KUKA KRL program: Wood_Test_2.src, Wood_Test_2.dat

--- Wood_Test_2.src ---
&ACCESS RVEO
&REL 38
&PARAM DISKPATH = KRC:\R1\Program\Milling
DEF Wood_Test_2 ( )
   INT lnActSt,lnUsedBase,lnActBase,lnUsedTool,lnBaseNr
   INT lnJobNr, lnCounter,lnCounter2
   FRAME lfZcut
   FRAME lfToolDiamShift
   FRAME lfStartMillingPos
   FRAME lfBaseShift
   FRAME lfBaseCycleZ
   FRAME lfBaseCycleShift

   CONTINUE
   ;IF ($T1 OR $T2)THEN
   GLOBAL INTERRUPT DECL 3 WHEN $STOPMESS==TRUE DO IR_STOPM ( )
   INTERRUPT ON 3
   BAS (#INITMOV,0)
   lnActSt = 1
   PTP $POS_ACT
   PTP lAstartPos

   gbRobControlActive = FALSE

   ; Used Base and tool
   lnUsedBase = 11
   lnActBase = 12
   lnUsedTool = 11

   gnLastToolNr = 5
   lnBaseNr = 23

   gfMillingOffset = $NULLFRAME

   lfZcut = $NULLFRAME
   lfZcut.Z = 0
   lfBaseShift = {X -30,Y -10,Z 1.1,A 0,B 0,C 0}
   lfBaseCycleZ = $NULLFRAME
   lfBaseCycleZ.Z = 0

   ;*************************************************************
   ;*                      Mill TOP SURFACE                     *
   ;*************************************************************
   grUsedRPM = GetMillingRPM(grTool_VC[gnLastToolNr], grTool_Diameter[gnLastToolNr])
   grUsedMillingSpeed = GetMillingSpeed(grUsedRPM, grTool_ToothCount[gnLastToolNr], grTool_FeedPerTooth[gnLastToolNr])

   SpindleRun(grUsedRPM,#CLOCKWISE)

   lfBaseCycleZ = $NULLFRAME
   lfBaseCycleZ.Z = 0
   BASE_DATA[lnUsedBase] = BASE_DATA[lnBaseNr] : lfBaseShift : lfBaseCycleZ
   TOOL_DATA[lnUsedTool] = TOOL_DATA[gnLastToolNr] :{X 0,Y 0,Z 0,A 270,B 0,C 0}

   MoveSettings(lnUsedBase, lnUsedTool, 100, grUsedMillingSpeed)
   ;; Move To PreposMillingPos Point P1 {5mm far from WP surface}
   lfToolDiamShift   = $NULLFRAME
   lfToolDiamShift.X = 0
   lfToolDiamShift.Y = 0
   lfToolDiamShift.Z = 5
   lfStartMillingPos = lfWorkPos[1] : lfToolDiamShift
   LIN lfStartMillingPos

   lfBaseCycleShift = $NULLFRAME
   BASE_DATA[lnActBase] = BASE_DATA[lnUsedBase]
   FOR lnCounter = 1 TO 2

      FOR lnCounter2 = 1 TO 2
         SWITCH lnCounter2
            CASE 1
               grUsedRPM = GetMillingRPM(grTool_VC[gnLastToolNr], grTool_Diameter[gnLastToolNr])
               grUsedMillingSpeed = GetMillingSpeed(grUsedRPM, grTool_ToothCount[gnLastToolNr], grTool_FeedPerTooth[gnLastToolNr])
            CASE 2
               grUsedRPM = GetMillingRPM(grTool_VC[gnLastToolNr], grTool_Diameter[gnLastToolNr])*1.5
               grUsedMillingSpeed = GetMillingSpeed(grUsedRPM, grTool_ToothCount[gnLastToolNr], grTool_FeedPerTooth[gnLastToolNr])/1.5
         ENDSWITCH
         SpindleRun(grUsedRPM,#CLOCKWISE)
         ;; Move To Milling Point P1
         MoveSettings(lnActBase, lnUsedTool, 100, grUsedMillingSpeed)
         lfToolDiamShift   =   $NULLFRAME
         lfToolDiamShift.x =  0
         lfToolDiamShift.Y =  0
         lfToolDiamShift.Z =   - (0.1 *lnCounter)
         LIN lfWorkPos[1]:lfToolDiamShift C_VEL

         ;; Move To Milling Point P2
         MoveSettings(lnActBase, lnUsedTool, 100, grUsedMillingSpeed)
         lfToolDiamShift   =   $NULLFRAME
         lfToolDiamShift.x =  0
         lfToolDiamShift.Y =  0
         lfToolDiamShift.Z =   - (0.1 *lnCounter)
         LIN lfWorkPos[2]:lfToolDiamShift C_VEL

         ;; Move To Milling Point P2
         MoveSettings(lnActBase, lnUsedTool, 100, grUsedMillingSpeed)
         lfToolDiamShift   =   $NULLFRAME
         lfToolDiamShift.x =  grTool_Diameter[gnLastToolNr] -1;* 2
         lfToolDiamShift.Y =  0
         lfToolDiamShift.Z =   - (0.1 *lnCounter)
         LIN lfWorkPos[2]:lfToolDiamShift C_VEL

         ;; Move To Milling Point P1
         MoveSettings(lnActBase, lnUsedTool, 100, grUsedMillingSpeed)
         lfToolDiamShift   =   $NULLFRAME
         lfToolDiamShift.x =  grTool_Diameter[gnLastToolNr] -1 ;* 2
         lfToolDiamShift.Y =  0
         lfToolDiamShift.Z =  - (0.1 *lnCounter)
         LIN lfWorkPos[1]:lfToolDiamShift C_VEL

         lfBaseCycleShift.X = lfBaseCycleShift.X +(grTool_Diameter[gnLastToolNr] * 2 )-1
         BASE_DATA[lnActBase] = BASE_DATA[lnUsedBase] : lfBaseCycleShift
      ENDFOR
      LIN_REL {Z 5} C_VEL #TOOL
      lfBaseCycleShift = $NULLFRAME
      lfBaseCycleShift.X = 0
      BASE_DATA[lnActBase] = BASE_DATA[lnUsedBase]
      MoveSettings(lnActBase, lnUsedTool, 100, grUsedMillingSpeed)
      ;; Move To PreposMillingPos Point P1 {5mm far from WP surface}
      lfToolDiamShift   = $NULLFRAME
      lfToolDiamShift.X = 0
      lfToolDiamShift.Y = 0
      lfToolDiamShift.Z = 5
      lfStartMillingPos = lfWorkPos[1] : lfToolDiamShift
      LIN lfStartMillingPos

   ENDFOR

   MoveSettings(lnUsedBase, lnUsedTool, 100, 500)
   ;; End of Milling Move Out of the WP
   TRIGGER WHEN DISTANCE=1 DELAY=0 DO  SpindleSetSpeed(50) PRIO=-1
   LIN_REL {Z 5} C_VEL #TOOL

   LIN_REL {Z 100} C_VEL #BASE

   TOOL_DATA[lnUsedTool] = TOOL_DATA[gnLastToolNr] :{X 0,Y 0,Z 0,A 180,B 90,C -90}
   MoveSettings(lnUsedBase, lnUsedTool, 100, 500)
   PTP lastartpos C_PTP

   WAIT SEC 1
   SpindleStop()

END

--- Wood_Test_2.dat ---
&ACCESS RVEO
&REL 38
&PARAM DISKPATH = KRC:\R1\Program\Milling
DEFDAT  WOOD_TEST_2 PUBLIC

DECL AXIS lAstartPos={A1 -22.4984303,A2 -99.5414124,A3 132.718292,A4 75.8801346,A5 -68.2717209,A6 -55.2195663}
DECL FRAME lfPrePos[5]
lfPrePos[1]={X -32.0000,Y -50.0000,Z 350.000,A 90.0000,B 0.0,C -45.0000}
lfPrePos[2]={X -32.0000,Y -15.0000,Z 70.0000,A 90.0000,B 0.0,C -90.0000}
lfPrePos[3]={X 0.0,Y -32.0000,Z 70.0000,A 0.0,B 0.0,C 90.0000}
lfPrePos[4]={X 0.0,Y -32.0000,Z 50.0000,A 90.0000,B 0.0,C 0.0}
lfPrePos[5]={X 0.0,Y -50.0000,Z 350.000,A 90.0000,B 0.0,C 0.0}

DECL FRAME lfWorkPos[12]
lfWorkPos[1]={X 0.0,Y 180.000,Z 0.0,A 0.0,B 0.0,C 0.0}
lfWorkPos[2]={X 0.0,Y -40.0,Z 0.0,A 0.0,B 0.0,C 0.0}
lfWorkPos[3]={X 0.0,Y 0.0,Z 0.0,A 0.0,B 0.0,C 90.0000}
lfWorkPos[4]={X 0.0,Y 200.000,Z 0.0,A 0.0,B 0.0,C 90.0000}

lfWorkPos[5]={X 12.5000,Y 340.000,Z 0.0,A 0.0,B 0.0,C 0.0}
lfWorkPos[6]={X 12.5000,Y 12.5000,Z 0.0,A 0.0,B 0.0,C 0.0}
lfWorkPos[7]={X 200.000,Y 12.5000,Z 0.0,A 0.0,B 0.0,C 0.0}

lfWorkPos[8]={X 200.000,Y 1.00000,Z 0.0,A 0.0,B 0.0,C 45.0000}
lfWorkPos[9]={X 0.0,Y 1.00000,Z 0.0,A 0.0,B 0.0,C 45.0000}
lfWorkPos[10]={X 1.00000,Y 0.0,Z 0.0,A 0.0,B -45.0000,C 0.0}
lfWorkPos[11]={X 1.00000,Y 200.000,Z 0.0,A 0.0,B -45.0000,C 0.0}
ENDDAT
